{attribute 'qualified_only'}
TYPE PLCopenStatusBase :
(
	ERR_OK := 0,
	ERROR := 1,	
	ABORTED := 2,	
	ENABLED_WAITING := 65533,	
	NOT_ENABLED := 65534,	
	BUSY := 65535	
);
END_TYPE

(* stored: Version 1.1.0.1
   EnumerationTextList PLCopenStatusBase: Id {affdcb97-526e-49da-8e66-616feef77d1f} *)
